// TIA Portal V20 export
DATA_BLOCK "CallUnit_DB"   // DB12
{ DB_Accessible_From_OPC_UA := 'FALSE' }
AUTHOR : ERsystem_FA2_DH. Kim
// stored: AssignedProDiagFB Unit1.ProDiag, DBAccessibleFromOPCUA false, DBAccessibleFromWebserver false, InstanceOfName Unit1.CallUnit, InstanceOfType FB, Namespace Unit1
"Unit1.CallUnit"
   // VAR_INPUT
   //    safetyReleased : Bool := TRUE;
   // END_VAR
   // VAR_OUTPUT
   //    acknowledgeSafety { ExternalWritable := 'False'} : Bool := FALSE;
   // END_VAR
   // VAR_IN_OUT
   //    globalStatus : "LAF_typeGeneralStatus";
   //    unitInterface : "LAF_typeUnitInterface";
   // END_VAR
   // VAR
   //    instManageAlarms { ExternalWritable := 'False'} : "LAF_ManageAlarms";
   //    instStatusCollector { ExternalWritable := 'False'} : "LUC_StatusCollector";
   //    instInterfaceManager { ExternalWritable := 'False'} : "LUC_InterfaceManager";
   //    instUnitModeStateManager { ExternalWritable := 'False'} : "LPMLV2022_UnitModeStateManager";
   //    instRemoteInterfaceOpcUa { ExternalWritable := 'False'} : "LUC_RemoteCtrl_OpcUa";
   //    instSignalStack { ExternalWritable := 'False'} : "LUC_SignalStack";
   //    instUnitModeStateTimes { ExternalWritable := 'False'} : "LPMLV2022_UnitModeStateTimes";
   //    instUnitModeChangeAllowed { ExternalWritable := 'False'} : "LPMLV2022_UnitModeChangeAllowed";
   //    instPFEEvents { S7_SetPoint := 'True'} : "Unit1.EventsPFE";
   //    statTonTime { S7_SetPoint := 'True'} : Array[0..99] of TON_TIME;
   //    instTofTimer { ExternalWritable := 'False'} : Array[0..9] of TOF_TIME;
   //    instEQP_Interface_BA010 { ExternalWritable := 'False'} : "LER_EQP_Interface_ReelCut";
   //    instEQP_Interface_BA015 { ExternalWritable := 'False'} : "LER_EQP_Interface_ReelCut";
   //    instEQP_Interface_BA060 { ExternalWritable := 'False'} : "LER_EQP_Interface_Inspection";
   //    instEQP_Interface_BA030 { ExternalWritable := 'False'} : "LER_EQP_Interface_OtherStack";
   //    BSEND_Instance_BA10 { S7_SetPoint := 'True'} : BSEND;
   //    BRCV_Instance_BA10 { S7_SetPoint := 'True'} : BRCV;
   //    BSEND_Instance_BA15 { S7_SetPoint := 'True'} : BSEND;
   //    BRCV_Instance_BA15 { S7_SetPoint := 'True'} : BRCV;
   //    BSEND_Instance_BA40 { S7_SetPoint := 'True'} : BSEND;
   //    BRCV_Instance_BA40 { S7_SetPoint := 'True'} : BRCV;
   //    BSEND_Instance_BA60 { S7_SetPoint := 'True'} : BSEND;
   //    BRCV_Instance_BA60 { S7_SetPoint := 'True'} : BRCV;
   //    instSinaInfeed { ExternalWritable := 'False'} : SinaInfeed;
   //    statRemoteInterface { ExternalWritable := 'False'} : "LUC_typeCommands";
   //    statLocalInterface { ExternalWritable := 'False'} : "LUC_typeCommands";
   //    statEmEnableCheck { ExternalWritable := 'False'} : Array[0..2] of Bool;
   //    statSpecialFuctionEnableCheck : Array[0..2] of Bool;
   //    statEmHomeScCheck { ExternalWritable := 'False'} : Array[0..7] of Bool;
   //    statPulse { ExternalWritable := 'False'} : Array[0..99] of Bool;
   //    statNoModeCmd { ExternalWritable := 'False'} : Bool;
   //    statEnableManualCmds : Bool;
   //    sleep { S7_SetPoint := 'True'} : "LER_typeSleepMode";
   //    statPreElectrodeNumber : Struct
   //       anode : DInt;
   //       cathode : DInt;
   //       currentTotalEL : DInt;
   //    END_STRUCT;
   //    instCalculateOut { S7_SetPoint := 'True'} : "LER_Calculate_Out";
   //    instStackMainCommand { S7_SetPoint := 'True'} : "LER_StackMainCommand";
   //    InstLER_FFU_LIU117 { S7_SetPoint := 'True'} : "LER_FFU_LIU117";
   //    sMotionToPLC { S7_SetPoint := 'True'} : "LER_typeCommonDataStackMotion";
   //    StatAllEmLinked { S7_SetPoint := 'True'} : Bool;
   //    citi_Ptrig : Array[0..20] of Bool;
   //    citiTon : Array[0..20] of TON_TIME;
   //    citi : Time;
   //    citiTest : Array[0..20] of Bool;
   //    statCalculateParameters : Struct
   //       AnodeCount : DInt;
   //       CathodeCount : DInt;
   //       SepaCount : DInt;
   //       TotalThickness : LReal;
   //       TotalSepaWebLenth : LReal;
   //    END_STRUCT;
   // END_VAR
BEGIN
   instManageAlarms.proDiagState.Total_Number := 562;
   instManageAlarms.proDiagState.All := FALSE;
   instManageAlarms.proDiagState.O := FALSE;
   instManageAlarms.proDiagState.I := FALSE;
   instManageAlarms.proDiagState.R := FALSE;
   instManageAlarms.proDiagState."A" := FALSE;
   instManageAlarms.proDiagState.P := FALSE;
   instManageAlarms.proDiagState.Merr := FALSE;
   instManageAlarms.proDiagState.Mtxt := FALSE;
   instManageAlarms.proDiagState.SV_Types := 16#00;
   instManageAlarms.proDiagState.C1 := FALSE;
   instManageAlarms.proDiagState.C2 := FALSE;
   instManageAlarms.proDiagState.C3 := FALSE;
   instManageAlarms.proDiagState.C4 := FALSE;
   instManageAlarms.proDiagState.C5 := FALSE;
   instManageAlarms.proDiagState.C6 := FALSE;
   instManageAlarms.proDiagState.C7 := FALSE;
   instManageAlarms.proDiagState.C8 := FALSE;
   instManageAlarms.proDiagState.Categories := 16#00;
   instManageAlarms.proDiagState.Sub_Cat_1 := 16#0000_0000;
   instManageAlarms.proDiagState.Sub_Cat_2 := 16#0000_0000;
   instManageAlarms.proDiagState.Reserved := 16#00;
   instManageAlarms.parentAlarmDB.error := FALSE;
   instManageAlarms.parentAlarmDB.warning := FALSE;
   instManageAlarms.parentAlarmDB.info := FALSE;
   instManageAlarms.alarmDB.error := FALSE;
   instManageAlarms.alarmDB.warning := FALSE;
   instManageAlarms.alarmDB.info := FALSE;
   instManageAlarms.hmiInterfaceDB.error := FALSE;
   instManageAlarms.hmiInterfaceDB.warning := FALSE;
   instManageAlarms.hmiInterfaceDB.info := FALSE;
   instInterfaceManager.processInterface.reset := FALSE;
   instInterfaceManager.processInterface.start := FALSE;
   instInterfaceManager.processInterface.stop := FALSE;
   instInterfaceManager.processInterface.hold := FALSE;
   instInterfaceManager.processInterface.unhold := FALSE;
   instInterfaceManager.processInterface.suspend := FALSE;
   instInterfaceManager.processInterface.unsuspend := FALSE;
   instInterfaceManager.processInterface.abort := FALSE;
   instInterfaceManager.processInterface.clear := FALSE;
   instInterfaceManager.processInterface.complete := FALSE;
   instInterfaceManager.processInterface.stateComplete := TRUE;
   instInterfaceManager.enableLocalInterface := TRUE;
   instInterfaceManager.localInterface.modeRequests.production := FALSE;
   instInterfaceManager.localInterface.modeRequests.maintenance := TRUE;
   instInterfaceManager.localInterface.modeRequests.manual := FALSE;
   instInterfaceManager.localInterface.modeRequests.nomode := FALSE;
   instInterfaceManager.localInterface.modeRequests.sleep := FALSE;
   instInterfaceManager.localInterface.modeRequests.deepsleep := FALSE;
   instInterfaceManager.localInterface.modeRequests.userMode04 := FALSE;
   instInterfaceManager.localInterface.modeRequests.userMode05 := FALSE;
   instInterfaceManager.localInterface.modeRequests.userMode06 := FALSE;
   instInterfaceManager.localInterface.modeRequests.userMode07 := FALSE;
   instInterfaceManager.localInterface.modeRequests.userMode08 := FALSE;
   instInterfaceManager.localInterface.modeRequests.userMode09 := FALSE;
   instInterfaceManager.localInterface.modeRequests.userMode10 := FALSE;
   instInterfaceManager.localInterface.modeRequests.userMode11 := FALSE;
   instInterfaceManager.localInterface.modeRequests.userMode12 := FALSE;
   instInterfaceManager.localInterface.modeRequests.userMode13 := FALSE;
   instInterfaceManager.localInterface.stateCommands.reset := FALSE;
   instInterfaceManager.localInterface.stateCommands.start := FALSE;
   instInterfaceManager.localInterface.stateCommands.stop := FALSE;
   instInterfaceManager.localInterface.stateCommands.hold := FALSE;
   instInterfaceManager.localInterface.stateCommands.unhold := FALSE;
   instInterfaceManager.localInterface.stateCommands.suspend := FALSE;
   instInterfaceManager.localInterface.stateCommands.unsuspend := FALSE;
   instInterfaceManager.localInterface.stateCommands.abort := FALSE;
   instInterfaceManager.localInterface.stateCommands.clear := FALSE;
   instInterfaceManager.localInterface.stateCommands.complete := FALSE;
   instInterfaceManager.localInterface.stateCommands.stateComplete := FALSE;
   instInterfaceManager.enableHmiInterface := FALSE;
   instInterfaceManager.hmiInterface.modeRequests.production := FALSE;
   instInterfaceManager.hmiInterface.modeRequests.maintenance := FALSE;
   instInterfaceManager.hmiInterface.modeRequests.manual := FALSE;
   instInterfaceManager.hmiInterface.modeRequests.nomode := FALSE;
   instInterfaceManager.hmiInterface.modeRequests.sleep := FALSE;
   instInterfaceManager.hmiInterface.modeRequests.deepsleep := FALSE;
   instInterfaceManager.hmiInterface.modeRequests.userMode04 := FALSE;
   instInterfaceManager.hmiInterface.modeRequests.userMode05 := FALSE;
   instInterfaceManager.hmiInterface.modeRequests.userMode06 := FALSE;
   instInterfaceManager.hmiInterface.modeRequests.userMode07 := FALSE;
   instInterfaceManager.hmiInterface.modeRequests.userMode08 := FALSE;
   instInterfaceManager.hmiInterface.modeRequests.userMode09 := FALSE;
   instInterfaceManager.hmiInterface.modeRequests.userMode10 := FALSE;
   instInterfaceManager.hmiInterface.modeRequests.userMode11 := FALSE;
   instInterfaceManager.hmiInterface.modeRequests.userMode12 := FALSE;
   instInterfaceManager.hmiInterface.modeRequests.userMode13 := FALSE;
   instInterfaceManager.hmiInterface.stateCommands.reset := FALSE;
   instInterfaceManager.hmiInterface.stateCommands.start := FALSE;
   instInterfaceManager.hmiInterface.stateCommands.stop := FALSE;
   instInterfaceManager.hmiInterface.stateCommands.hold := FALSE;
   instInterfaceManager.hmiInterface.stateCommands.unhold := FALSE;
   instInterfaceManager.hmiInterface.stateCommands.suspend := FALSE;
   instInterfaceManager.hmiInterface.stateCommands.unsuspend := FALSE;
   instInterfaceManager.hmiInterface.stateCommands.abort := FALSE;
   instInterfaceManager.hmiInterface.stateCommands.clear := FALSE;
   instInterfaceManager.hmiInterface.stateCommands.complete := FALSE;
   instInterfaceManager.hmiInterface.stateCommands.stateComplete := FALSE;
   instInterfaceManager.enableRemoteInterface := FALSE;
   instInterfaceManager.remoteInterface.modeRequests.production := FALSE;
   instInterfaceManager.remoteInterface.modeRequests.maintenance := FALSE;
   instInterfaceManager.remoteInterface.modeRequests.manual := FALSE;
   instInterfaceManager.remoteInterface.modeRequests.nomode := FALSE;
   instInterfaceManager.remoteInterface.modeRequests.sleep := FALSE;
   instInterfaceManager.remoteInterface.modeRequests.deepsleep := FALSE;
   instInterfaceManager.remoteInterface.modeRequests.userMode04 := FALSE;
   instInterfaceManager.remoteInterface.modeRequests.userMode05 := FALSE;
   instInterfaceManager.remoteInterface.modeRequests.userMode06 := FALSE;
   instInterfaceManager.remoteInterface.modeRequests.userMode07 := FALSE;
   instInterfaceManager.remoteInterface.modeRequests.userMode08 := FALSE;
   instInterfaceManager.remoteInterface.modeRequests.userMode09 := FALSE;
   instInterfaceManager.remoteInterface.modeRequests.userMode10 := FALSE;
   instInterfaceManager.remoteInterface.modeRequests.userMode11 := FALSE;
   instInterfaceManager.remoteInterface.modeRequests.userMode12 := FALSE;
   instInterfaceManager.remoteInterface.modeRequests.userMode13 := FALSE;
   instInterfaceManager.remoteInterface.stateCommands.reset := FALSE;
   instInterfaceManager.remoteInterface.stateCommands.start := FALSE;
   instInterfaceManager.remoteInterface.stateCommands.stop := FALSE;
   instInterfaceManager.remoteInterface.stateCommands.hold := FALSE;
   instInterfaceManager.remoteInterface.stateCommands.unhold := FALSE;
   instInterfaceManager.remoteInterface.stateCommands.suspend := FALSE;
   instInterfaceManager.remoteInterface.stateCommands.unsuspend := FALSE;
   instInterfaceManager.remoteInterface.stateCommands.abort := FALSE;
   instInterfaceManager.remoteInterface.stateCommands.clear := FALSE;
   instInterfaceManager.remoteInterface.stateCommands.complete := FALSE;
   instInterfaceManager.remoteInterface.stateCommands.stateComplete := FALSE;
   instInterfaceManager.unitMode := 0;
   instInterfaceManager.unitModeChangeRequest := FALSE;
   instInterfaceManager.cntrlCmd := 3;
   instInterfaceManager.cmdChangeRequest := FALSE;
   instInterfaceManager.SC := FALSE;
   instInterfaceManager.localControlEnabled := TRUE;
   instInterfaceManager.hmiControlEnabled := FALSE;
   instInterfaceManager.remoteControlEnabled := FALSE;
   instInterfaceManager.error := FALSE;
   instInterfaceManager.status := 16#0000;
   instInterfaceManager.statRequested.mode := 0;
   instInterfaceManager.statRequested.state := 0;
   instInterfaceManager.statPrevious.modesLocalInterface := 16#0002;
   instInterfaceManager.statPrevious.modesRemoteInterface := 16#0000;
   instInterfaceManager.statPrevious.modesHmiInterface := 16#0000;
   instInterfaceManager.statPrevious.statesProcessInterface := 16#0400;
   instInterfaceManager.statPrevious.statesLocalInterface := 16#0000;
   instInterfaceManager.statPrevious.statesRemoteInterface := 16#0000;
   instInterfaceManager.statPrevious.statesHmiInterface := 16#0000;
   instInterfaceManager.statStatus := 16#0000;
   instUnitModeStateManager.UnitMode := 0;
   instUnitModeStateManager.UnitModeChangeRequest := FALSE;
   instUnitModeStateManager.CntrlCmd := 3;
   instUnitModeStateManager.CmdChangeRequest := FALSE;
   instUnitModeStateManager.SC := FALSE;
   instUnitModeStateManager.configuration.EnabledModesCfg := 16#0000_001E;
   instUnitModeStateManager.configuration.DisabledStatesCfg[0..1] := 16#0000_0000;
   instUnitModeStateManager.configuration.DisabledStatesCfg[2] := 16#0003_6020;
   instUnitModeStateManager.configuration.DisabledStatesCfg[3] := 16#0003_7C28;
   instUnitModeStateManager.configuration.DisabledStatesCfg[4..16] := 16#0000_0000;
   instUnitModeStateManager.configuration.ModeTransitionCfg[0..16] := 16#0000_0214;
   instUnitModeStateManager.configuration.holdCmdCfg := 16#0000_0040;
   instUnitModeStateManager.configuration.completeCmdCfg := 16#0000_0860;
   instUnitModeStateManager.UnitModeCurrent := 2;
   instUnitModeStateManager.StateCurrent := 2;
   instUnitModeStateManager.StateRequested := 2;
   instUnitModeStateManager.StateChangeInProcess := FALSE;
   instUnitModeStateManager.CurDisabledStates := 16#0003_6020;
   instUnitModeStateManager.curHoldCmdCfg := 16#0000_0040;
   instUnitModeStateManager.curCompleteCmdCfg := 16#0000_0000;
   instUnitModeStateManager.unitModeChangeNotAllowed := FALSE;
   instUnitModeStateManager.cntrlCmdNotAllowed := FALSE;
   instUnitModeStateManager.diagnostics.bufferIndex := 7;
   instUnitModeStateManager.diagnostics.buffer[0].timestamp := DTL#2026-01-06-06:46:51.371465172;
   instUnitModeStateManager.diagnostics.buffer[1].timestamp := DTL#2026-01-06-06:46:51.374585015;
   instUnitModeStateManager.diagnostics.buffer[2].timestamp := DTL#2026-01-06-06:46:51.567016868;
   instUnitModeStateManager.diagnostics.buffer[3].timestamp := DTL#2026-01-06-06:46:55.878705971;
   instUnitModeStateManager.diagnostics.buffer[4].timestamp := DTL#2026-01-06-06:46:55.971592245;
   instUnitModeStateManager.diagnostics.buffer[5].timestamp := DTL#2026-01-06-06:46:58.882031211;
   instUnitModeStateManager.diagnostics.buffer[6].timestamp := DTL#2026-01-06-06:46:58.884831167;
   instUnitModeStateManager.diagnostics.buffer[7].timestamp := DTL#2026-01-06-06:46:58.887783077;
   instUnitModeStateManager.diagnostics.buffer[0..2].UnitModeCurrent := 2;
   instUnitModeStateManager.diagnostics.buffer[3..6].UnitModeCurrent := 4;
   instUnitModeStateManager.diagnostics.buffer[7].UnitModeCurrent := 2;
   instUnitModeStateManager.diagnostics.buffer[0].StateCurrent := 8;
   instUnitModeStateManager.diagnostics.buffer[1..3].StateCurrent := 9;
   instUnitModeStateManager.diagnostics.buffer[4..5].StateCurrent := 1;
   instUnitModeStateManager.diagnostics.buffer[6..7].StateCurrent := 2;
   instUnitModeStateManager.diagnostics.buffer[0].UnitMode := 0;
   instUnitModeStateManager.diagnostics.buffer[1].UnitMode := 2;
   instUnitModeStateManager.diagnostics.buffer[2].UnitMode := 4;
   instUnitModeStateManager.diagnostics.buffer[3..5].UnitMode := 0;
   instUnitModeStateManager.diagnostics.buffer[6].UnitMode := 2;
   instUnitModeStateManager.diagnostics.buffer[7].UnitMode := 0;
   instUnitModeStateManager.diagnostics.buffer[0..2].CntrlCmd := 8;
   instUnitModeStateManager.diagnostics.buffer[3].CntrlCmd := 9;
   instUnitModeStateManager.diagnostics.buffer[4..7].CntrlCmd := 3;
   instUnitModeStateManager.diagnostics.buffer[0].SC := TRUE;
   instUnitModeStateManager.diagnostics.buffer[1..4].SC := FALSE;
   instUnitModeStateManager.diagnostics.buffer[5].SC := TRUE;
   instUnitModeStateManager.diagnostics.buffer[6].SC := FALSE;
   instUnitModeStateManager.diagnostics.buffer[7].SC := TRUE;
   instUnitModeStateManager.diagnostics.buffer[0].message := 16#02;
   instUnitModeStateManager.diagnostics.buffer[1].message := 16#03;
   instUnitModeStateManager.diagnostics.buffer[2].message := 16#01;
   instUnitModeStateManager.diagnostics.buffer[3].message := 16#02;
   instUnitModeStateManager.diagnostics.buffer[4].message := 16#84;
   instUnitModeStateManager.diagnostics.buffer[5].message := 16#02;
   instUnitModeStateManager.diagnostics.buffer[6].message := 16#01;
   instUnitModeStateManager.diagnostics.buffer[7].message := 16#85;
   instUnitModeStateManager.statConfiguration.EnabledModesCfg := 16#0000_001E;
   instUnitModeStateManager.statConfiguration.DisabledStatesCfg[0..1] := 16#0000_0000;
   instUnitModeStateManager.statConfiguration.DisabledStatesCfg[2] := 16#0003_6020;
   instUnitModeStateManager.statConfiguration.DisabledStatesCfg[3] := 16#0003_7C28;
   instUnitModeStateManager.statConfiguration.DisabledStatesCfg[4] := 16#000FFFFF;
   instUnitModeStateManager.statConfiguration.DisabledStatesCfg[5..16] := 16#0000_0000;
   instUnitModeStateManager.statConfiguration.ModeTransitionCfg[0..16] := 16#0000_0214;
   instUnitModeStateManager.statConfiguration.holdCmdCfg := 16#0000_0040;
   instUnitModeStateManager.statConfiguration.completeCmdCfg := 16#0000_0860;
   instUnitModeStateManager.statUnitModeChangeRequest := FALSE;
   instUnitModeStateManager.statCmdChangeRequest := FALSE;
   instUnitModeStateManager.statFirstCycle := FALSE;
   instUnitModeStateManager.statSCOld := FALSE;
   instUnitModeStateManager.statUnitMode := 0;
   instUnitModeStateManager.statUnitModeOld := 0;
   instUnitModeStateManager.statUnitModeCurrentInternal := 2;
   instUnitModeStateManager.statUnitModeCurrentInternalOld := 0;
   instUnitModeStateManager.statStateCurrentOld := 2;
   instUnitModeStateManager.statStateInternal := 2;
   instUnitModeStateManager.statStateInternalOld := 0;
   instUnitModeStateManager.statCntrlCmdOld := 0;
   instUnitModeStateManager.statStatesInCurrentMode.clearing := TRUE;
   instUnitModeStateManager.statStatesInCurrentMode.stopped := TRUE;
   instUnitModeStateManager.statStatesInCurrentMode.starting := TRUE;
   instUnitModeStateManager.statStatesInCurrentMode.idle := TRUE;
   instUnitModeStateManager.statStatesInCurrentMode.suspended := FALSE;
   instUnitModeStateManager.statStatesInCurrentMode.execute := TRUE;
   instUnitModeStateManager.statStatesInCurrentMode.stopping := TRUE;
   instUnitModeStateManager.statStatesInCurrentMode.aborting := TRUE;
   instUnitModeStateManager.statStatesInCurrentMode.aborted := TRUE;
   instUnitModeStateManager.statStatesInCurrentMode.holding := TRUE;
   instUnitModeStateManager.statStatesInCurrentMode.held := TRUE;
   instUnitModeStateManager.statStatesInCurrentMode.unholding := TRUE;
   instUnitModeStateManager.statStatesInCurrentMode.suspending := FALSE;
   instUnitModeStateManager.statStatesInCurrentMode.unsuspending := FALSE;
   instUnitModeStateManager.statStatesInCurrentMode.resetting := TRUE;
   instUnitModeStateManager.statStatesInCurrentMode.completing := FALSE;
   instUnitModeStateManager.statStatesInCurrentMode.completed := FALSE;
   instUnitModeStateManager.statConsiderHoldCmdIn.starting := FALSE;
   instUnitModeStateManager.statConsiderHoldCmdIn.idle := FALSE;
   instUnitModeStateManager.statConsiderHoldCmdIn.suspended := FALSE;
   instUnitModeStateManager.statConsiderHoldCmdIn.execute := TRUE;
   instUnitModeStateManager.statConsiderHoldCmdIn.unholding := FALSE;
   instUnitModeStateManager.statConsiderHoldCmdIn.suspending := FALSE;
   instUnitModeStateManager.statConsiderHoldCmdIn.unsuspending := FALSE;
   instUnitModeStateManager.statConsiderHoldCmdIn.completing := FALSE;
   instUnitModeStateManager.statConsiderHoldCmdIn.completed := FALSE;
   instUnitModeStateManager.statConsiderCompleteCmdIn.suspended := FALSE;
   instUnitModeStateManager.statConsiderCompleteCmdIn.execute := FALSE;
   instUnitModeStateManager.statConsiderCompleteCmdIn.held := FALSE;
   instUnitModeStateManager.statCmdChangeRequestOld := FALSE;
   instUnitModeStateManager.statUnitModeChangeRequestOld := FALSE;
   instUnitModeStateManager.statDiagnosticsBufferIndex := 7;
   instUnitModeStateManager.statStateRequested := 2;
   instUnitModeStateManager.statUnitModeChangeNotAllowed := FALSE;
   instUnitModeStateManager.statCntrlCmdNotAllowed := FALSE;
   instRemoteInterfaceOpcUa.remoteControlEnabled := FALSE;
   instRemoteInterfaceOpcUa.currentState := 2;
   instRemoteInterfaceOpcUa.currentMode := 2;
   instRemoteInterfaceOpcUa.cntrlCmdDenied := FALSE;
   instRemoteInterfaceOpcUa.unitModeChangeNotAllowed := FALSE;
   instRemoteInterfaceOpcUa.configuration.enableMethods.reset := TRUE;
   instRemoteInterfaceOpcUa.configuration.enableMethods.start := TRUE;
   instRemoteInterfaceOpcUa.configuration.enableMethods.stop := TRUE;
   instRemoteInterfaceOpcUa.configuration.enableMethods.hold := TRUE;
   instRemoteInterfaceOpcUa.configuration.enableMethods.unhold := TRUE;
   instRemoteInterfaceOpcUa.configuration.enableMethods.suspend := TRUE;
   instRemoteInterfaceOpcUa.configuration.enableMethods.unsuspend := TRUE;
   instRemoteInterfaceOpcUa.configuration.enableMethods.abort := TRUE;
   instRemoteInterfaceOpcUa.configuration.enableMethods.clear := TRUE;
   instRemoteInterfaceOpcUa.configuration.enableMethods.complete := TRUE;
   instRemoteInterfaceOpcUa.configuration.enableMethods.stateComplete := TRUE;
   instRemoteInterfaceOpcUa.configuration.enableMethods.requestUnitMode := TRUE;
   instRemoteInterfaceOpcUa.configuration.enableMethods.requestUnitState := TRUE;
   instRemoteInterfaceOpcUa.error := FALSE;
   instRemoteInterfaceOpcUa.status := 16#0000;
   instRemoteInterfaceOpcUa.subfunctionStatus := 16#0000_0000;
   instRemoteInterfaceOpcUa.instReset.methodEnable := TRUE;
   instRemoteInterfaceOpcUa.instReset.remoteControlEnabled := FALSE;
   instRemoteInterfaceOpcUa.instReset.currentState := 2;
   instRemoteInterfaceOpcUa.instReset.cntrlCmdDenied := FALSE;
   instRemoteInterfaceOpcUa.instReset.error := FALSE;
   instRemoteInterfaceOpcUa.instReset.status := 16#7000;
   instRemoteInterfaceOpcUa.instReset.subfunctionStatus := 16#0000_0000;
   instRemoteInterfaceOpcUa.instReset.OPC_UA_ServerMethodPre_Instance.Done := FALSE;
   instRemoteInterfaceOpcUa.instReset.OPC_UA_ServerMethodPre_Instance.Busy := FALSE;
   instRemoteInterfaceOpcUa.instReset.OPC_UA_ServerMethodPre_Instance.Error := FALSE;
   instRemoteInterfaceOpcUa.instReset.OPC_UA_ServerMethodPre_Instance.Status := 16#0070_0000;
   instRemoteInterfaceOpcUa.instReset.OPC_UA_ServerMethodPre_Instance.UAMethod_Called := FALSE;
   instRemoteInterfaceOpcUa.instReset.OPC_UA_ServerMethodPost_Instance.UAMethod_Result := 16#0000_0000;
   instRemoteInterfaceOpcUa.instReset.OPC_UA_ServerMethodPost_Instance.UAMethod_Finished := FALSE;
   instRemoteInterfaceOpcUa.instReset.OPC_UA_ServerMethodPost_Instance.Done := FALSE;
   instRemoteInterfaceOpcUa.instReset.OPC_UA_ServerMethodPost_Instance.Busy := FALSE;
   instRemoteInterfaceOpcUa.instReset.OPC_UA_ServerMethodPost_Instance.Error := FALSE;
   instRemoteInterfaceOpcUa.instReset.OPC_UA_ServerMethodPost_Instance.Status := 16#0070_0000;
   instRemoteInterfaceOpcUa.instStart.methodEnable := TRUE;
   instRemoteInterfaceOpcUa.instStart.remoteControlEnabled := FALSE;
   instRemoteInterfaceOpcUa.instStart.currentState := 2;
   instRemoteInterfaceOpcUa.instStart.cntrlCmdDenied := FALSE;
   instRemoteInterfaceOpcUa.instStart.error := FALSE;
   instRemoteInterfaceOpcUa.instStart.status := 16#7000;
   instRemoteInterfaceOpcUa.instStart.subfunctionStatus := 16#0000_0000;
   instRemoteInterfaceOpcUa.instStart.OPC_UA_ServerMethodPre_Instance.Done := FALSE;
   instRemoteInterfaceOpcUa.instStart.OPC_UA_ServerMethodPre_Instance.Busy := FALSE;
   instRemoteInterfaceOpcUa.instStart.OPC_UA_ServerMethodPre_Instance.Error := FALSE;
   instRemoteInterfaceOpcUa.instStart.OPC_UA_ServerMethodPre_Instance.Status := 16#0070_0000;
   instRemoteInterfaceOpcUa.instStart.OPC_UA_ServerMethodPre_Instance.UAMethod_Called := FALSE;
   instRemoteInterfaceOpcUa.instStart.OPC_UA_ServerMethodPost_Instance.UAMethod_Result := 16#0000_0000;
   instRemoteInterfaceOpcUa.instStart.OPC_UA_ServerMethodPost_Instance.UAMethod_Finished := FALSE;
   instRemoteInterfaceOpcUa.instStart.OPC_UA_ServerMethodPost_Instance.Done := FALSE;
   instRemoteInterfaceOpcUa.instStart.OPC_UA_ServerMethodPost_Instance.Busy := FALSE;
   instRemoteInterfaceOpcUa.instStart.OPC_UA_ServerMethodPost_Instance.Error := FALSE;
   instRemoteInterfaceOpcUa.instStart.OPC_UA_ServerMethodPost_Instance.Status := 16#0070_0000;
   instRemoteInterfaceOpcUa.instStop.methodEnable := TRUE;
   instRemoteInterfaceOpcUa.instStop.remoteControlEnabled := FALSE;
   instRemoteInterfaceOpcUa.instStop.currentState := 2;
   instRemoteInterfaceOpcUa.instStop.cntrlCmdDenied := FALSE;
   instRemoteInterfaceOpcUa.instStop.error := FALSE;
   instRemoteInterfaceOpcUa.instStop.status := 16#7000;
   instRemoteInterfaceOpcUa.instStop.subfunctionStatus := 16#0000_0000;
   instRemoteInterfaceOpcUa.instStop.OPC_UA_ServerMethodPre_Instance.Done := FALSE;
   instRemoteInterfaceOpcUa.instStop.OPC_UA_ServerMethodPre_Instance.Busy := FALSE;
   instRemoteInterfaceOpcUa.instStop.OPC_UA_ServerMethodPre_Instance.Error := FALSE;
   instRemoteInterfaceOpcUa.instStop.OPC_UA_ServerMethodPre_Instance.Status := 16#0070_0000;
   instRemoteInterfaceOpcUa.instStop.OPC_UA_ServerMethodPre_Instance.UAMethod_Called := FALSE;
   instRemoteInterfaceOpcUa.instStop.OPC_UA_ServerMethodPost_Instance.UAMethod_Result := 16#0000_0000;
   instRemoteInterfaceOpcUa.instStop.OPC_UA_ServerMethodPost_Instance.UAMethod_Finished := FALSE;
   instRemoteInterfaceOpcUa.instStop.OPC_UA_ServerMethodPost_Instance.Done := FALSE;
   instRemoteInterfaceOpcUa.instStop.OPC_UA_ServerMethodPost_Instance.Busy := FALSE;
   instRemoteInterfaceOpcUa.instStop.OPC_UA_ServerMethodPost_Instance.Error := FALSE;
   instRemoteInterfaceOpcUa.instStop.OPC_UA_ServerMethodPost_Instance.Status := 16#0070_0000;
   instRemoteInterfaceOpcUa.instHold.methodEnable := TRUE;
   instRemoteInterfaceOpcUa.instHold.remoteControlEnabled := FALSE;
   instRemoteInterfaceOpcUa.instHold.currentState := 2;
   instRemoteInterfaceOpcUa.instHold.cntrlCmdDenied := FALSE;
   instRemoteInterfaceOpcUa.instHold.error := FALSE;
   instRemoteInterfaceOpcUa.instHold.status := 16#7000;
   instRemoteInterfaceOpcUa.instHold.subfunctionStatus := 16#0000_0000;
   instRemoteInterfaceOpcUa.instHold.OPC_UA_ServerMethodPre_Instance.Done := FALSE;
   instRemoteInterfaceOpcUa.instHold.OPC_UA_ServerMethodPre_Instance.Busy := FALSE;
   instRemoteInterfaceOpcUa.instHold.OPC_UA_ServerMethodPre_Instance.Error := FALSE;
   instRemoteInterfaceOpcUa.instHold.OPC_UA_ServerMethodPre_Instance.Status := 16#0070_0000;
   instRemoteInterfaceOpcUa.instHold.OPC_UA_ServerMethodPre_Instance.UAMethod_Called := FALSE;
   instRemoteInterfaceOpcUa.instHold.OPC_UA_ServerMethodPost_Instance.UAMethod_Result := 16#0000_0000;
   instRemoteInterfaceOpcUa.instHold.OPC_UA_ServerMethodPost_Instance.UAMethod_Finished := FALSE;
   instRemoteInterfaceOpcUa.instHold.OPC_UA_ServerMethodPost_Instance.Done := FALSE;
   instRemoteInterfaceOpcUa.instHold.OPC_UA_ServerMethodPost_Instance.Busy := FALSE;
   instRemoteInterfaceOpcUa.instHold.OPC_UA_ServerMethodPost_Instance.Error := FALSE;
   instRemoteInterfaceOpcUa.instHold.OPC_UA_ServerMethodPost_Instance.Status := 16#0070_0000;
   instRemoteInterfaceOpcUa.instUnhold.methodEnable := TRUE;
   instRemoteInterfaceOpcUa.instUnhold.remoteControlEnabled := FALSE;
   instRemoteInterfaceOpcUa.instUnhold.currentState := 2;
   instRemoteInterfaceOpcUa.instUnhold.cntrlCmdDenied := FALSE;
   instRemoteInterfaceOpcUa.instUnhold.error := FALSE;
   instRemoteInterfaceOpcUa.instUnhold.status := 16#7000;
   instRemoteInterfaceOpcUa.instUnhold.subfunctionStatus := 16#0000_0000;
   instRemoteInterfaceOpcUa.instUnhold.OPC_UA_ServerMethodPre_Instance.Done := FALSE;
   instRemoteInterfaceOpcUa.instUnhold.OPC_UA_ServerMethodPre_Instance.Busy := FALSE;
   instRemoteInterfaceOpcUa.instUnhold.OPC_UA_ServerMethodPre_Instance.Error := FALSE;
   instRemoteInterfaceOpcUa.instUnhold.OPC_UA_ServerMethodPre_Instance.Status := 16#0070_0000;
   instRemoteInterfaceOpcUa.instUnhold.OPC_UA_ServerMethodPre_Instance.UAMethod_Called := FALSE;
   instRemoteInterfaceOpcUa.instUnhold.OPC_UA_ServerMethodPost_Instance.UAMethod_Result := 16#0000_0000;
   instRemoteInterfaceOpcUa.instUnhold.OPC_UA_ServerMethodPost_Instance.UAMethod_Finished := FALSE;
   instRemoteInterfaceOpcUa.instUnhold.OPC_UA_ServerMethodPost_Instance.Done := FALSE;
   instRemoteInterfaceOpcUa.instUnhold.OPC_UA_ServerMethodPost_Instance.Busy := FALSE;
   instRemoteInterfaceOpcUa.instUnhold.OPC_UA_ServerMethodPost_Instance.Error := FALSE;
   instRemoteInterfaceOpcUa.instUnhold.OPC_UA_ServerMethodPost_Instance.Status := 16#0070_0000;
   instRemoteInterfaceOpcUa.instSuspend.methodEnable := TRUE;
   instRemoteInterfaceOpcUa.instSuspend.remoteControlEnabled := FALSE;
   instRemoteInterfaceOpcUa.instSuspend.currentState := 2;
   instRemoteInterfaceOpcUa.instSuspend.cntrlCmdDenied := FALSE;
   instRemoteInterfaceOpcUa.instSuspend.error := FALSE;
   instRemoteInterfaceOpcUa.instSuspend.status := 16#7000;
   instRemoteInterfaceOpcUa.instSuspend.subfunctionStatus := 16#0000_0000;
   instRemoteInterfaceOpcUa.instSuspend.OPC_UA_ServerMethodPre_Instance.Done := FALSE;
   instRemoteInterfaceOpcUa.instSuspend.OPC_UA_ServerMethodPre_Instance.Busy := FALSE;
   instRemoteInterfaceOpcUa.instSuspend.OPC_UA_ServerMethodPre_Instance.Error := FALSE;
   instRemoteInterfaceOpcUa.instSuspend.OPC_UA_ServerMethodPre_Instance.Status := 16#0070_0000;
   instRemoteInterfaceOpcUa.instSuspend.OPC_UA_ServerMethodPre_Instance.UAMethod_Called := FALSE;
   instRemoteInterfaceOpcUa.instSuspend.OPC_UA_ServerMethodPost_Instance.UAMethod_Result := 16#0000_0000;
   instRemoteInterfaceOpcUa.instSuspend.OPC_UA_ServerMethodPost_Instance.UAMethod_Finished := FALSE;
   instRemoteInterfaceOpcUa.instSuspend.OPC_UA_ServerMethodPost_Instance.Done := FALSE;
   instRemoteInterfaceOpcUa.instSuspend.OPC_UA_ServerMethodPost_Instance.Busy := FALSE;
   instRemoteInterfaceOpcUa.instSuspend.OPC_UA_ServerMethodPost_Instance.Error := FALSE;
   instRemoteInterfaceOpcUa.instSuspend.OPC_UA_ServerMethodPost_Instance.Status := 16#0070_0000;
   instRemoteInterfaceOpcUa.instUnsuspend.methodEnable := TRUE;
   instRemoteInterfaceOpcUa.instUnsuspend.remoteControlEnabled := FALSE;
   instRemoteInterfaceOpcUa.instUnsuspend.currentState := 2;
   instRemoteInterfaceOpcUa.instUnsuspend.cntrlCmdDenied := FALSE;
   instRemoteInterfaceOpcUa.instUnsuspend.error := FALSE;
   instRemoteInterfaceOpcUa.instUnsuspend.status := 16#7000;
   instRemoteInterfaceOpcUa.instUnsuspend.subfunctionStatus := 16#0000_0000;
   instRemoteInterfaceOpcUa.instUnsuspend.OPC_UA_ServerMethodPre_Instance.Done := FALSE;
   instRemoteInterfaceOpcUa.instUnsuspend.OPC_UA_ServerMethodPre_Instance.Busy := FALSE;
   instRemoteInterfaceOpcUa.instUnsuspend.OPC_UA_ServerMethodPre_Instance.Error := FALSE;
   instRemoteInterfaceOpcUa.instUnsuspend.OPC_UA_ServerMethodPre_Instance.Status := 16#0070_0000;
   instRemoteInterfaceOpcUa.instUnsuspend.OPC_UA_ServerMethodPre_Instance.UAMethod_Called := FALSE;
   instRemoteInterfaceOpcUa.instUnsuspend.OPC_UA_ServerMethodPost_Instance.UAMethod_Result := 16#0000_0000;
   instRemoteInterfaceOpcUa.instUnsuspend.OPC_UA_ServerMethodPost_Instance.UAMethod_Finished := FALSE;
   instRemoteInterfaceOpcUa.instUnsuspend.OPC_UA_ServerMethodPost_Instance.Done := FALSE;
   instRemoteInterfaceOpcUa.instUnsuspend.OPC_UA_ServerMethodPost_Instance.Busy := FALSE;
   instRemoteInterfaceOpcUa.instUnsuspend.OPC_UA_ServerMethodPost_Instance.Error := FALSE;
   instRemoteInterfaceOpcUa.instUnsuspend.OPC_UA_ServerMethodPost_Instance.Status := 16#0070_0000;
   instRemoteInterfaceOpcUa.instAbort.methodEnable := TRUE;
   instRemoteInterfaceOpcUa.instAbort.remoteControlEnabled := FALSE;
   instRemoteInterfaceOpcUa.instAbort.currentState := 2;
   instRemoteInterfaceOpcUa.instAbort.cntrlCmdDenied := FALSE;
   instRemoteInterfaceOpcUa.instAbort.error := FALSE;
   instRemoteInterfaceOpcUa.instAbort.status := 16#7000;
   instRemoteInterfaceOpcUa.instAbort.subfunctionStatus := 16#0000_0000;
   instRemoteInterfaceOpcUa.instAbort.OPC_UA_ServerMethodPre_Instance.Done := FALSE;
   instRemoteInterfaceOpcUa.instAbort.OPC_UA_ServerMethodPre_Instance.Busy := FALSE;
   instRemoteInterfaceOpcUa.instAbort.OPC_UA_ServerMethodPre_Instance.Error := FALSE;
   instRemoteInterfaceOpcUa.instAbort.OPC_UA_ServerMethodPre_Instance.Status := 16#0070_0000;
   instRemoteInterfaceOpcUa.instAbort.OPC_UA_ServerMethodPre_Instance.UAMethod_Called := FALSE;
   instRemoteInterfaceOpcUa.instAbort.OPC_UA_ServerMethodPost_Instance.UAMethod_Result := 16#0000_0000;
   instRemoteInterfaceOpcUa.instAbort.OPC_UA_ServerMethodPost_Instance.UAMethod_Finished := FALSE;
   instRemoteInterfaceOpcUa.instAbort.OPC_UA_ServerMethodPost_Instance.Done := FALSE;
   instRemoteInterfaceOpcUa.instAbort.OPC_UA_ServerMethodPost_Instance.Busy := FALSE;
   instRemoteInterfaceOpcUa.instAbort.OPC_UA_ServerMethodPost_Instance.Error := FALSE;
   instRemoteInterfaceOpcUa.instAbort.OPC_UA_ServerMethodPost_Instance.Status := 16#0070_0000;
   instRemoteInterfaceOpcUa.instClear.methodEnable := TRUE;
   instRemoteInterfaceOpcUa.instClear.remoteControlEnabled := FALSE;
   instRemoteInterfaceOpcUa.instClear.currentState := 2;
   instRemoteInterfaceOpcUa.instClear.cntrlCmdDenied := FALSE;
   instRemoteInterfaceOpcUa.instClear.error := FALSE;
   instRemoteInterfaceOpcUa.instClear.status := 16#7000;
   instRemoteInterfaceOpcUa.instClear.subfunctionStatus := 16#0000_0000;
   instRemoteInterfaceOpcUa.instClear.OPC_UA_ServerMethodPre_Instance.Done := FALSE;
   instRemoteInterfaceOpcUa.instClear.OPC_UA_ServerMethodPre_Instance.Busy := FALSE;
   instRemoteInterfaceOpcUa.instClear.OPC_UA_ServerMethodPre_Instance.Error := FALSE;
   instRemoteInterfaceOpcUa.instClear.OPC_UA_ServerMethodPre_Instance.Status := 16#0070_0000;
   instRemoteInterfaceOpcUa.instClear.OPC_UA_ServerMethodPre_Instance.UAMethod_Called := FALSE;
   instRemoteInterfaceOpcUa.instClear.OPC_UA_ServerMethodPost_Instance.UAMethod_Result := 16#0000_0000;
   instRemoteInterfaceOpcUa.instClear.OPC_UA_ServerMethodPost_Instance.UAMethod_Finished := FALSE;
   instRemoteInterfaceOpcUa.instClear.OPC_UA_ServerMethodPost_Instance.Done := FALSE;
   instRemoteInterfaceOpcUa.instClear.OPC_UA_ServerMethodPost_Instance.Busy := FALSE;
   instRemoteInterfaceOpcUa.instClear.OPC_UA_ServerMethodPost_Instance.Error := FALSE;
   instRemoteInterfaceOpcUa.instClear.OPC_UA_ServerMethodPost_Instance.Status := 16#0070_0000;
   instRemoteInterfaceOpcUa.instComplete.methodEnable := TRUE;
   instRemoteInterfaceOpcUa.instComplete.remoteControlEnabled := FALSE;
   instRemoteInterfaceOpcUa.instComplete.currentState := 2;
   instRemoteInterfaceOpcUa.instComplete.cntrlCmdDenied := FALSE;
   instRemoteInterfaceOpcUa.instComplete.error := FALSE;
   instRemoteInterfaceOpcUa.instComplete.status := 16#7000;
   instRemoteInterfaceOpcUa.instComplete.subfunctionStatus := 16#0000_0000;
   instRemoteInterfaceOpcUa.instComplete.OPC_UA_ServerMethodPre_Instance.Done := FALSE;
   instRemoteInterfaceOpcUa.instComplete.OPC_UA_ServerMethodPre_Instance.Busy := FALSE;
   instRemoteInterfaceOpcUa.instComplete.OPC_UA_ServerMethodPre_Instance.Error := FALSE;
   instRemoteInterfaceOpcUa.instComplete.OPC_UA_ServerMethodPre_Instance.Status := 16#0070_0000;
   instRemoteInterfaceOpcUa.instComplete.OPC_UA_ServerMethodPre_Instance.UAMethod_Called := FALSE;
   instRemoteInterfaceOpcUa.instComplete.OPC_UA_ServerMethodPost_Instance.UAMethod_Result := 16#0000_0000;
   instRemoteInterfaceOpcUa.instComplete.OPC_UA_ServerMethodPost_Instance.UAMethod_Finished := FALSE;
   instRemoteInterfaceOpcUa.instComplete.OPC_UA_ServerMethodPost_Instance.Done := FALSE;
   instRemoteInterfaceOpcUa.instComplete.OPC_UA_ServerMethodPost_Instance.Busy := FALSE;
   instRemoteInterfaceOpcUa.instComplete.OPC_UA_ServerMethodPost_Instance.Error := FALSE;
   instRemoteInterfaceOpcUa.instComplete.OPC_UA_ServerMethodPost_Instance.Status := 16#0070_0000;
   instRemoteInterfaceOpcUa.instStateComplete.methodEnable := TRUE;
   instRemoteInterfaceOpcUa.instStateComplete.remoteControlEnabled := FALSE;
   instRemoteInterfaceOpcUa.instStateComplete.currentState := 2;
   instRemoteInterfaceOpcUa.instStateComplete.cntrlCmdDenied := FALSE;
   instRemoteInterfaceOpcUa.instStateComplete.error := FALSE;
   instRemoteInterfaceOpcUa.instStateComplete.status := 16#7000;
   instRemoteInterfaceOpcUa.instStateComplete.subfunctionStatus := 16#0000_0000;
   instRemoteInterfaceOpcUa.instStateComplete.OPC_UA_ServerMethodPre_Instance.Done := FALSE;
   instRemoteInterfaceOpcUa.instStateComplete.OPC_UA_ServerMethodPre_Instance.Busy := FALSE;
   instRemoteInterfaceOpcUa.instStateComplete.OPC_UA_ServerMethodPre_Instance.Error := FALSE;
   instRemoteInterfaceOpcUa.instStateComplete.OPC_UA_ServerMethodPre_Instance.Status := 16#0070_0000;
   instRemoteInterfaceOpcUa.instStateComplete.OPC_UA_ServerMethodPre_Instance.UAMethod_Called := FALSE;
   instRemoteInterfaceOpcUa.instStateComplete.OPC_UA_ServerMethodPost_Instance.UAMethod_Result := 16#0000_0000;
   instRemoteInterfaceOpcUa.instStateComplete.OPC_UA_ServerMethodPost_Instance.UAMethod_Finished := FALSE;
   instRemoteInterfaceOpcUa.instStateComplete.OPC_UA_ServerMethodPost_Instance.Done := FALSE;
   instRemoteInterfaceOpcUa.instStateComplete.OPC_UA_ServerMethodPost_Instance.Busy := FALSE;
   instRemoteInterfaceOpcUa.instStateComplete.OPC_UA_ServerMethodPost_Instance.Error := FALSE;
   instRemoteInterfaceOpcUa.instStateComplete.OPC_UA_ServerMethodPost_Instance.Status := 16#0070_0000;
   instRemoteInterfaceOpcUa.instSetUnitMode.methodEnable := TRUE;
   instRemoteInterfaceOpcUa.instSetUnitMode.remoteControlEnabled := FALSE;
   instRemoteInterfaceOpcUa.instSetUnitMode.currentMode := 2;
   instRemoteInterfaceOpcUa.instSetUnitMode.unitModeChangeDenied := FALSE;
   instRemoteInterfaceOpcUa.instSetUnitMode.error := FALSE;
   instRemoteInterfaceOpcUa.instSetUnitMode.status := 16#7000;
   instRemoteInterfaceOpcUa.instSetUnitMode.subfunctionStatus := 16#0000_0000;
   instRemoteInterfaceOpcUa.instSetUnitMode.OPC_UA_ServerMethodPre_Instance.Done := FALSE;
   instRemoteInterfaceOpcUa.instSetUnitMode.OPC_UA_ServerMethodPre_Instance.Busy := FALSE;
   instRemoteInterfaceOpcUa.instSetUnitMode.OPC_UA_ServerMethodPre_Instance.Error := FALSE;
   instRemoteInterfaceOpcUa.instSetUnitMode.OPC_UA_ServerMethodPre_Instance.Status := 16#0070_0000;
   instRemoteInterfaceOpcUa.instSetUnitMode.OPC_UA_ServerMethodPre_Instance.UAMethod_Called := FALSE;
   instRemoteInterfaceOpcUa.instSetUnitMode.OPC_UA_ServerMethodPost_Instance.UAMethod_Result := 16#0000_0000;
   instRemoteInterfaceOpcUa.instSetUnitMode.OPC_UA_ServerMethodPost_Instance.UAMethod_Finished := FALSE;
   instRemoteInterfaceOpcUa.instSetUnitMode.OPC_UA_ServerMethodPost_Instance.Done := FALSE;
   instRemoteInterfaceOpcUa.instSetUnitMode.OPC_UA_ServerMethodPost_Instance.Busy := FALSE;
   instRemoteInterfaceOpcUa.instSetUnitMode.OPC_UA_ServerMethodPost_Instance.Error := FALSE;
   instRemoteInterfaceOpcUa.instSetUnitMode.OPC_UA_ServerMethodPost_Instance.Status := 16#0070_0000;
   instRemoteInterfaceOpcUa.instSetUnitMode.UAMethod_InParameters.RequestedMode := 0;
   instRemoteInterfaceOpcUa.instSetUnitMode.statLastCycleMode := 2;
   instRemoteInterfaceOpcUa.instSetUnitState.methodEnable := TRUE;
   instRemoteInterfaceOpcUa.instSetUnitState.remoteControlEnabled := FALSE;
   instRemoteInterfaceOpcUa.instSetUnitState.currentState := 2;
   instRemoteInterfaceOpcUa.instSetUnitState.cntrlCmdDenied := FALSE;
   instRemoteInterfaceOpcUa.instSetUnitState.error := FALSE;
   instRemoteInterfaceOpcUa.instSetUnitState.status := 16#7000;
   instRemoteInterfaceOpcUa.instSetUnitState.subfunctionStatus := 16#0000_0000;
   instRemoteInterfaceOpcUa.instSetUnitState.OPC_UA_ServerMethodPre_Instance.Done := FALSE;
   instRemoteInterfaceOpcUa.instSetUnitState.OPC_UA_ServerMethodPre_Instance.Busy := FALSE;
   instRemoteInterfaceOpcUa.instSetUnitState.OPC_UA_ServerMethodPre_Instance.Error := FALSE;
   instRemoteInterfaceOpcUa.instSetUnitState.OPC_UA_ServerMethodPre_Instance.Status := 16#0070_0000;
   instRemoteInterfaceOpcUa.instSetUnitState.OPC_UA_ServerMethodPre_Instance.UAMethod_Called := FALSE;
   instRemoteInterfaceOpcUa.instSetUnitState.OPC_UA_ServerMethodPost_Instance.UAMethod_Result := 16#0000_0000;
   instRemoteInterfaceOpcUa.instSetUnitState.OPC_UA_ServerMethodPost_Instance.UAMethod_Finished := FALSE;
   instRemoteInterfaceOpcUa.instSetUnitState.OPC_UA_ServerMethodPost_Instance.Done := FALSE;
   instRemoteInterfaceOpcUa.instSetUnitState.OPC_UA_ServerMethodPost_Instance.Busy := FALSE;
   instRemoteInterfaceOpcUa.instSetUnitState.OPC_UA_ServerMethodPost_Instance.Error := FALSE;
   instRemoteInterfaceOpcUa.instSetUnitState.OPC_UA_ServerMethodPost_Instance.Status := 16#0070_0000;
   instRemoteInterfaceOpcUa.instSetUnitState.UAMethod_InParameters.RequestedCommand := 0;
   instRemoteInterfaceOpcUa.instSetUnitState.statLastCycleState := 2;
   instSignalStack.currentState := 0;
   instSignalStack.freqClockBit := FALSE;
   instSignalStack.disableHorn := FALSE;
   instSignalStack.hornPulseTime := T#0MS;
   instSignalStack.processBypass.static.red := FALSE;
   instSignalStack.processBypass.static.yellow := FALSE;
   instSignalStack.processBypass.static.blue := FALSE;
   instSignalStack.processBypass.static.green := FALSE;
   instSignalStack.processBypass.static.horn := FALSE;
   instSignalStack.processBypass.static.white := FALSE;
   instSignalStack.processBypass.static.user1 := FALSE;
   instSignalStack.processBypass.static.user2 := FALSE;
   instSignalStack.processBypass.flashing.red := FALSE;
   instSignalStack.processBypass.flashing.yellow := FALSE;
   instSignalStack.processBypass.flashing.blue := FALSE;
   instSignalStack.processBypass.flashing.green := FALSE;
   instSignalStack.processBypass.flashing.horn := FALSE;
   instSignalStack.processBypass.flashing.white := FALSE;
   instSignalStack.processBypass.flashing.user1 := FALSE;
   instSignalStack.processBypass.flashing.user2 := FALSE;
   instSignalStack.configuration.undefined.static.red := FALSE;
   instSignalStack.configuration.undefined.static.yellow := FALSE;
   instSignalStack.configuration.undefined.static.blue := FALSE;
   instSignalStack.configuration.undefined.static.green := FALSE;
   instSignalStack.configuration.undefined.static.horn := FALSE;
   instSignalStack.configuration.undefined.static.white := FALSE;
   instSignalStack.configuration.undefined.static.user1 := FALSE;
   instSignalStack.configuration.undefined.static.user2 := FALSE;
   instSignalStack.configuration.undefined.flashing.red := TRUE;
   instSignalStack.configuration.undefined.flashing.yellow := FALSE;
   instSignalStack.configuration.undefined.flashing.blue := FALSE;
   instSignalStack.configuration.undefined.flashing.green := FALSE;
   instSignalStack.configuration.undefined.flashing.horn := FALSE;
   instSignalStack.configuration.undefined.flashing.white := FALSE;
   instSignalStack.configuration.undefined.flashing.user1 := FALSE;
   instSignalStack.configuration.undefined.flashing.user2 := FALSE;
   instSignalStack.configuration.clearing.static.red := FALSE;
   instSignalStack.configuration.clearing.static.yellow := FALSE;
   instSignalStack.configuration.clearing.static.blue := FALSE;
   instSignalStack.configuration.clearing.static.green := FALSE;
   instSignalStack.configuration.clearing.static.horn := FALSE;
   instSignalStack.configuration.clearing.static.white := FALSE;
   instSignalStack.configuration.clearing.static.user1 := FALSE;
   instSignalStack.configuration.clearing.static.user2 := FALSE;
   instSignalStack.configuration.clearing.flashing.red := TRUE;
   instSignalStack.configuration.clearing.flashing.yellow := FALSE;
   instSignalStack.configuration.clearing.flashing.blue := FALSE;
   instSignalStack.configuration.clearing.flashing.green := FALSE;
   instSignalStack.configuration.clearing.flashing.horn := FALSE;
   instSignalStack.configuration.clearing.flashing.white := FALSE;
   instSignalStack.configuration.clearing.flashing.user1 := FALSE;
   instSignalStack.configuration.clearing.flashing.user2 := FALSE;
   instSignalStack.configuration.stopped.static.red := TRUE;
   instSignalStack.configuration.stopped.static.yellow := FALSE;
   instSignalStack.configuration.stopped.static.blue := FALSE;
   instSignalStack.configuration.stopped.static.green := FALSE;
   instSignalStack.configuration.stopped.static.horn := FALSE;
   instSignalStack.configuration.stopped.static.white := FALSE;
   instSignalStack.configuration.stopped.static.user1 := FALSE;
   instSignalStack.configuration.stopped.static.user2 := FALSE;
   instSignalStack.configuration.stopped.flashing.red := FALSE;
   instSignalStack.configuration.stopped.flashing.yellow := FALSE;
   instSignalStack.configuration.stopped.flashing.blue := FALSE;
   instSignalStack.configuration.stopped.flashing.green := FALSE;
   instSignalStack.configuration.stopped.flashing.horn := FALSE;
   instSignalStack.configuration.stopped.flashing.white := FALSE;
   instSignalStack.configuration.stopped.flashing.user1 := FALSE;
   instSignalStack.configuration.stopped.flashing.user2 := FALSE;
   instSignalStack.configuration.starting.static.red := FALSE;
   instSignalStack.configuration.starting.static.yellow := FALSE;
   instSignalStack.configuration.starting.static.blue := FALSE;
   instSignalStack.configuration.starting.static.green := TRUE;
   instSignalStack.configuration.starting.static.horn := FALSE;
   instSignalStack.configuration.starting.static.white := FALSE;
   instSignalStack.configuration.starting.static.user1 := FALSE;
   instSignalStack.configuration.starting.static.user2 := FALSE;
   instSignalStack.configuration.starting.flashing.red := FALSE;
   instSignalStack.configuration.starting.flashing.yellow := FALSE;
   instSignalStack.configuration.starting.flashing.blue := FALSE;
   instSignalStack.configuration.starting.flashing.green := FALSE;
   instSignalStack.configuration.starting.flashing.horn := FALSE;
   instSignalStack.configuration.starting.flashing.white := FALSE;
   instSignalStack.configuration.starting.flashing.user1 := FALSE;
   instSignalStack.configuration.starting.flashing.user2 := FALSE;
   instSignalStack.configuration.idle.static.red := FALSE;
   instSignalStack.configuration.idle.static.yellow := FALSE;
   instSignalStack.configuration.idle.static.blue := FALSE;
   instSignalStack.configuration.idle.static.green := FALSE;
   instSignalStack.configuration.idle.static.horn := FALSE;
   instSignalStack.configuration.idle.static.white := FALSE;
   instSignalStack.configuration.idle.static.user1 := FALSE;
   instSignalStack.configuration.idle.static.user2 := FALSE;
   instSignalStack.configuration.idle.flashing.red := FALSE;
   instSignalStack.configuration.idle.flashing.yellow := FALSE;
   instSignalStack.configuration.idle.flashing.blue := FALSE;
   instSignalStack.configuration.idle.flashing.green := TRUE;
   instSignalStack.configuration.idle.flashing.horn := FALSE;
   instSignalStack.configuration.idle.flashing.white := FALSE;
   instSignalStack.configuration.idle.flashing.user1 := FALSE;
   instSignalStack.configuration.idle.flashing.user2 := FALSE;
   instSignalStack.configuration.suspended.static.red := FALSE;
   instSignalStack.configuration.suspended.static.yellow := TRUE;
   instSignalStack.configuration.suspended.static.blue := FALSE;
   instSignalStack.configuration.suspended.static.green := FALSE;
   instSignalStack.configuration.suspended.static.horn := FALSE;
   instSignalStack.configuration.suspended.static.white := FALSE;
   instSignalStack.configuration.suspended.static.user1 := FALSE;
   instSignalStack.configuration.suspended.static.user2 := FALSE;
   instSignalStack.configuration.suspended.flashing.red := FALSE;
   instSignalStack.configuration.suspended.flashing.yellow := FALSE;
   instSignalStack.configuration.suspended.flashing.blue := FALSE;
   instSignalStack.configuration.suspended.flashing.green := FALSE;
   instSignalStack.configuration.suspended.flashing.horn := FALSE;
   instSignalStack.configuration.suspended.flashing.white := FALSE;
   instSignalStack.configuration.suspended.flashing.user1 := FALSE;
   instSignalStack.configuration.suspended.flashing.user2 := FALSE;
   instSignalStack.configuration.execute.static.red := FALSE;
   instSignalStack.configuration.execute.static.yellow := FALSE;
   instSignalStack.configuration.execute.static.blue := FALSE;
   instSignalStack.configuration.execute.static.green := TRUE;
   instSignalStack.configuration.execute.static.horn := FALSE;
   instSignalStack.configuration.execute.static.white := FALSE;
   instSignalStack.configuration.execute.static.user1 := FALSE;
   instSignalStack.configuration.execute.static.user2 := FALSE;
   instSignalStack.configuration.execute.flashing.red := FALSE;
   instSignalStack.configuration.execute.flashing.yellow := FALSE;
   instSignalStack.configuration.execute.flashing.blue := FALSE;
   instSignalStack.configuration.execute.flashing.green := FALSE;
   instSignalStack.configuration.execute.flashing.horn := FALSE;
   instSignalStack.configuration.execute.flashing.white := FALSE;
   instSignalStack.configuration.execute.flashing.user1 := FALSE;
   instSignalStack.configuration.execute.flashing.user2 := FALSE;
   instSignalStack.configuration.stopping.static.red := TRUE;
   instSignalStack.configuration.stopping.static.yellow := FALSE;
   instSignalStack.configuration.stopping.static.blue := FALSE;
   instSignalStack.configuration.stopping.static.green := FALSE;
   instSignalStack.configuration.stopping.static.horn := FALSE;
   instSignalStack.configuration.stopping.static.white := FALSE;
   instSignalStack.configuration.stopping.static.user1 := FALSE;
   instSignalStack.configuration.stopping.static.user2 := FALSE;
   instSignalStack.configuration.stopping.flashing.red := FALSE;
   instSignalStack.configuration.stopping.flashing.yellow := FALSE;
   instSignalStack.configuration.stopping.flashing.blue := FALSE;
   instSignalStack.configuration.stopping.flashing.green := FALSE;
   instSignalStack.configuration.stopping.flashing.horn := FALSE;
   instSignalStack.configuration.stopping.flashing.white := FALSE;
   instSignalStack.configuration.stopping.flashing.user1 := FALSE;
   instSignalStack.configuration.stopping.flashing.user2 := FALSE;
   instSignalStack.configuration.aborting.static.red := FALSE;
   instSignalStack.configuration.aborting.static.yellow := FALSE;
   instSignalStack.configuration.aborting.static.blue := FALSE;
   instSignalStack.configuration.aborting.static.green := FALSE;
   instSignalStack.configuration.aborting.static.horn := FALSE;
   instSignalStack.configuration.aborting.static.white := FALSE;
   instSignalStack.configuration.aborting.static.user1 := FALSE;
   instSignalStack.configuration.aborting.static.user2 := FALSE;
   instSignalStack.configuration.aborting.flashing.red := TRUE;
   instSignalStack.configuration.aborting.flashing.yellow := FALSE;
   instSignalStack.configuration.aborting.flashing.blue := FALSE;
   instSignalStack.configuration.aborting.flashing.green := FALSE;
   instSignalStack.configuration.aborting.flashing.horn := FALSE;
   instSignalStack.configuration.aborting.flashing.white := FALSE;
   instSignalStack.configuration.aborting.flashing.user1 := FALSE;
   instSignalStack.configuration.aborting.flashing.user2 := FALSE;
   instSignalStack.configuration.aborted.static.red := FALSE;
   instSignalStack.configuration.aborted.static.yellow := FALSE;
   instSignalStack.configuration.aborted.static.blue := FALSE;
   instSignalStack.configuration.aborted.static.green := FALSE;
   instSignalStack.configuration.aborted.static.horn := FALSE;
   instSignalStack.configuration.aborted.static.white := FALSE;
   instSignalStack.configuration.aborted.static.user1 := FALSE;
   instSignalStack.configuration.aborted.static.user2 := FALSE;
   instSignalStack.configuration.aborted.flashing.red := TRUE;
   instSignalStack.configuration.aborted.flashing.yellow := FALSE;
   instSignalStack.configuration.aborted.flashing.blue := FALSE;
   instSignalStack.configuration.aborted.flashing.green := FALSE;
   instSignalStack.configuration.aborted.flashing.horn := FALSE;
   instSignalStack.configuration.aborted.flashing.white := FALSE;
   instSignalStack.configuration.aborted.flashing.user1 := FALSE;
   instSignalStack.configuration.aborted.flashing.user2 := FALSE;
   instSignalStack.configuration.holding.static.red := FALSE;
   instSignalStack.configuration.holding.static.yellow := FALSE;
   instSignalStack.configuration.holding.static.blue := FALSE;
   instSignalStack.configuration.holding.static.green := FALSE;
   instSignalStack.configuration.holding.static.horn := FALSE;
   instSignalStack.configuration.holding.static.white := FALSE;
   instSignalStack.configuration.holding.static.user1 := FALSE;
   instSignalStack.configuration.holding.static.user2 := FALSE;
   instSignalStack.configuration.holding.flashing.red := FALSE;
   instSignalStack.configuration.holding.flashing.yellow := FALSE;
   instSignalStack.configuration.holding.flashing.blue := TRUE;
   instSignalStack.configuration.holding.flashing.green := FALSE;
   instSignalStack.configuration.holding.flashing.horn := FALSE;
   instSignalStack.configuration.holding.flashing.white := FALSE;
   instSignalStack.configuration.holding.flashing.user1 := FALSE;
   instSignalStack.configuration.holding.flashing.user2 := FALSE;
   instSignalStack.configuration.held.static.red := FALSE;
   instSignalStack.configuration.held.static.yellow := FALSE;
   instSignalStack.configuration.held.static.blue := TRUE;
   instSignalStack.configuration.held.static.green := FALSE;
   instSignalStack.configuration.held.static.horn := FALSE;
   instSignalStack.configuration.held.static.white := FALSE;
   instSignalStack.configuration.held.static.user1 := FALSE;
   instSignalStack.configuration.held.static.user2 := FALSE;
   instSignalStack.configuration.held.flashing.red := FALSE;
   instSignalStack.configuration.held.flashing.yellow := FALSE;
   instSignalStack.configuration.held.flashing.blue := FALSE;
   instSignalStack.configuration.held.flashing.green := FALSE;
   instSignalStack.configuration.held.flashing.horn := FALSE;
   instSignalStack.configuration.held.flashing.white := FALSE;
   instSignalStack.configuration.held.flashing.user1 := FALSE;
   instSignalStack.configuration.held.flashing.user2 := FALSE;
   instSignalStack.configuration.unholding.static.red := FALSE;
   instSignalStack.configuration.unholding.static.yellow := FALSE;
   instSignalStack.configuration.unholding.static.blue := FALSE;
   instSignalStack.configuration.unholding.static.green := TRUE;
   instSignalStack.configuration.unholding.static.horn := FALSE;
   instSignalStack.configuration.unholding.static.white := FALSE;
   instSignalStack.configuration.unholding.static.user1 := FALSE;
   instSignalStack.configuration.unholding.static.user2 := FALSE;
   instSignalStack.configuration.unholding.flashing.red := FALSE;
   instSignalStack.configuration.unholding.flashing.yellow := FALSE;
   instSignalStack.configuration.unholding.flashing.blue := FALSE;
   instSignalStack.configuration.unholding.flashing.green := FALSE;
   instSignalStack.configuration.unholding.flashing.horn := FALSE;
   instSignalStack.configuration.unholding.flashing.white := FALSE;
   instSignalStack.configuration.unholding.flashing.user1 := FALSE;
   instSignalStack.configuration.unholding.flashing.user2 := FALSE;
   instSignalStack.configuration.suspending.static.red := FALSE;
   instSignalStack.configuration.suspending.static.yellow := FALSE;
   instSignalStack.configuration.suspending.static.blue := FALSE;
   instSignalStack.configuration.suspending.static.green := FALSE;
   instSignalStack.configuration.suspending.static.horn := FALSE;
   instSignalStack.configuration.suspending.static.white := FALSE;
   instSignalStack.configuration.suspending.static.user1 := FALSE;
   instSignalStack.configuration.suspending.static.user2 := FALSE;
   instSignalStack.configuration.suspending.flashing.red := FALSE;
   instSignalStack.configuration.suspending.flashing.yellow := TRUE;
   instSignalStack.configuration.suspending.flashing.blue := FALSE;
   instSignalStack.configuration.suspending.flashing.green := FALSE;
   instSignalStack.configuration.suspending.flashing.horn := FALSE;
   instSignalStack.configuration.suspending.flashing.white := FALSE;
   instSignalStack.configuration.suspending.flashing.user1 := FALSE;
   instSignalStack.configuration.suspending.flashing.user2 := FALSE;
   instSignalStack.configuration.unsuspending.static.red := FALSE;
   instSignalStack.configuration.unsuspending.static.yellow := FALSE;
   instSignalStack.configuration.unsuspending.static.blue := FALSE;
   instSignalStack.configuration.unsuspending.static.green := TRUE;
   instSignalStack.configuration.unsuspending.static.horn := FALSE;
   instSignalStack.configuration.unsuspending.static.white := FALSE;
   instSignalStack.configuration.unsuspending.static.user1 := FALSE;
   instSignalStack.configuration.unsuspending.static.user2 := FALSE;
   instSignalStack.configuration.unsuspending.flashing.red := FALSE;
   instSignalStack.configuration.unsuspending.flashing.yellow := FALSE;
   instSignalStack.configuration.unsuspending.flashing.blue := FALSE;
   instSignalStack.configuration.unsuspending.flashing.green := FALSE;
   instSignalStack.configuration.unsuspending.flashing.horn := FALSE;
   instSignalStack.configuration.unsuspending.flashing.white := FALSE;
   instSignalStack.configuration.unsuspending.flashing.user1 := FALSE;
   instSignalStack.configuration.unsuspending.flashing.user2 := FALSE;
   instSignalStack.configuration.resetting.static.red := TRUE;
   instSignalStack.configuration.resetting.static.yellow := FALSE;
   instSignalStack.configuration.resetting.static.blue := FALSE;
   instSignalStack.configuration.resetting.static.green := FALSE;
   instSignalStack.configuration.resetting.static.horn := FALSE;
   instSignalStack.configuration.resetting.static.white := FALSE;
   instSignalStack.configuration.resetting.static.user1 := FALSE;
   instSignalStack.configuration.resetting.static.user2 := FALSE;
   instSignalStack.configuration.resetting.flashing.red := FALSE;
   instSignalStack.configuration.resetting.flashing.yellow := FALSE;
   instSignalStack.configuration.resetting.flashing.blue := FALSE;
   instSignalStack.configuration.resetting.flashing.green := FALSE;
   instSignalStack.configuration.resetting.flashing.horn := FALSE;
   instSignalStack.configuration.resetting.flashing.white := FALSE;
   instSignalStack.configuration.resetting.flashing.user1 := FALSE;
   instSignalStack.configuration.resetting.flashing.user2 := FALSE;
   instSignalStack.configuration.completing.static.red := FALSE;
   instSignalStack.configuration.completing.static.yellow := FALSE;
   instSignalStack.configuration.completing.static.blue := FALSE;
   instSignalStack.configuration.completing.static.green := TRUE;
   instSignalStack.configuration.completing.static.horn := FALSE;
   instSignalStack.configuration.completing.static.white := FALSE;
   instSignalStack.configuration.completing.static.user1 := FALSE;
   instSignalStack.configuration.completing.static.user2 := FALSE;
   instSignalStack.configuration.completing.flashing.red := FALSE;
   instSignalStack.configuration.completing.flashing.yellow := FALSE;
   instSignalStack.configuration.completing.flashing.blue := FALSE;
   instSignalStack.configuration.completing.flashing.green := FALSE;
   instSignalStack.configuration.completing.flashing.horn := FALSE;
   instSignalStack.configuration.completing.flashing.white := FALSE;
   instSignalStack.configuration.completing.flashing.user1 := FALSE;
   instSignalStack.configuration.completing.flashing.user2 := FALSE;
   instSignalStack.configuration.completed.static.red := TRUE;
   instSignalStack.configuration.completed.static.yellow := FALSE;
   instSignalStack.configuration.completed.static.blue := FALSE;
   instSignalStack.configuration.completed.static.green := FALSE;
   instSignalStack.configuration.completed.static.horn := FALSE;
   instSignalStack.configuration.completed.static.white := FALSE;
   instSignalStack.configuration.completed.static.user1 := FALSE;
   instSignalStack.configuration.completed.static.user2 := FALSE;
   instSignalStack.configuration.completed.flashing.red := FALSE;
   instSignalStack.configuration.completed.flashing.yellow := FALSE;
   instSignalStack.configuration.completed.flashing.blue := FALSE;
   instSignalStack.configuration.completed.flashing.green := FALSE;
   instSignalStack.configuration.completed.flashing.horn := FALSE;
   instSignalStack.configuration.completed.flashing.white := FALSE;
   instSignalStack.configuration.completed.flashing.user1 := FALSE;
   instSignalStack.configuration.completed.flashing.user2 := FALSE;
   instSignalStack.lightsByBool.redSolid := FALSE;
   instSignalStack.lightsByBool.redFlashing := FALSE;
   instSignalStack.lightsByBool.yellowSolid := FALSE;
   instSignalStack.lightsByBool.yellowFlashing := FALSE;
   instSignalStack.lightsByBool.blueSolid := FALSE;
   instSignalStack.lightsByBool.blueFlashing := FALSE;
   instSignalStack.lightsByBool.greenSolid := FALSE;
   instSignalStack.lightsByBool.greenFlashing := FALSE;
   instSignalStack.lightsByBool.hornSolid := FALSE;
   instSignalStack.lightsByBool.hornFlashing := FALSE;
   instSignalStack.lightsByBool.whiteSolid := FALSE;
   instSignalStack.lightsByBool.whiteFlashing := FALSE;
   instSignalStack.lightsByBool.user1Solid := FALSE;
   instSignalStack.lightsByBool.user1Flashing := FALSE;
   instSignalStack.lightsByBool.user2Solid := FALSE;
   instSignalStack.lightsByBool.user2Flashing := FALSE;
   instSignalStack.lightsByDint.red := 0;
   instSignalStack.lightsByDint.yellow := 0;
   instSignalStack.lightsByDint.blue := 0;
   instSignalStack.lightsByDint.green := 0;
   instSignalStack.lightsByDint.horn := 0;
   instSignalStack.lightsByDint.white := 0;
   instSignalStack.lightsByDint.user1 := 0;
   instSignalStack.lightsByDint.user2 := 0;
   instSignalStack.lightsByDWord.statusByDWord := 16#0000_0000;
   instSignalStack.lightsStatus.red := FALSE;
   instSignalStack.lightsStatus.yellow := FALSE;
   instSignalStack.lightsStatus.blue := FALSE;
   instSignalStack.lightsStatus.green := FALSE;
   instSignalStack.lightsStatus.horn := FALSE;
   instSignalStack.lightsStatus.white := FALSE;
   instSignalStack.lightsStatus.user1 := FALSE;
   instSignalStack.lightsStatus.user2 := FALSE;
   instSignalStack.instPulseHorn.PT := T#1S;
   instSignalStack.instPulseHorn.IN := FALSE;
   instUnitModeStateTimes.UnitModeCurrent := 2;
   instUnitModeStateTimes.StateCurrent := 2;
   instUnitModeStateTimes.resetTimes := FALSE;
   instUnitModeStateTimes.ModeTimeCurrent := 47401;
   instUnitModeStateTimes.StateTimeCurrent := 47401;
   instUnitModeStateTimes.AccTimeSinceReset := 71237;
   instUnitModeStateTimes.actualTimeAllModes[0..1] := 0;
   instUnitModeStateTimes.actualTimeAllModes[2] := 47401;
   instUnitModeStateTimes.actualTimeAllModes[3] := 0;
   instUnitModeStateTimes.actualTimeAllModes[4] := 8;
   instUnitModeStateTimes.actualTimeAllModes[5..16] := 0;
   instUnitModeStateTimes.cumulativeTimeAllModes[0..1] := 0;
   instUnitModeStateTimes.cumulativeTimeAllModes[2] := 67801;
   instUnitModeStateTimes.cumulativeTimeAllModes[3] := 0;
   instUnitModeStateTimes.cumulativeTimeAllModes[4] := 3436;
   instUnitModeStateTimes.cumulativeTimeAllModes[5..16] := 0;
   instUnitModeStateTimes.actualTimeAllStatesOfAllModes[0,0..17] := 0;
   instUnitModeStateTimes.actualTimeAllStatesOfAllModes[1,0..17] := 0;
   instUnitModeStateTimes.actualTimeAllStatesOfAllModes[2,0] := 0;
   instUnitModeStateTimes.actualTimeAllStatesOfAllModes[2,1] := 3;
   instUnitModeStateTimes.actualTimeAllStatesOfAllModes[2,2] := 47401;
   instUnitModeStateTimes.actualTimeAllStatesOfAllModes[2,3..17] := 0;
   instUnitModeStateTimes.actualTimeAllStatesOfAllModes[3,0..17] := 0;
   instUnitModeStateTimes.actualTimeAllStatesOfAllModes[4,0] := 0;
   instUnitModeStateTimes.actualTimeAllStatesOfAllModes[4,1] := 3;
   instUnitModeStateTimes.actualTimeAllStatesOfAllModes[4,2..8] := 0;
   instUnitModeStateTimes.actualTimeAllStatesOfAllModes[4,9] := 5;
   instUnitModeStateTimes.actualTimeAllStatesOfAllModes[4,10..17] := 0;
   instUnitModeStateTimes.actualTimeAllStatesOfAllModes[5,0..17] := 0;
   instUnitModeStateTimes.actualTimeAllStatesOfAllModes[6,0..17] := 0;
   instUnitModeStateTimes.actualTimeAllStatesOfAllModes[7,0..17] := 0;
   instUnitModeStateTimes.actualTimeAllStatesOfAllModes[8,0..17] := 0;
   instUnitModeStateTimes.actualTimeAllStatesOfAllModes[9,0..17] := 0;
   instUnitModeStateTimes.actualTimeAllStatesOfAllModes[10,0..17] := 0;
   instUnitModeStateTimes.actualTimeAllStatesOfAllModes[11,0..17] := 0;
   instUnitModeStateTimes.actualTimeAllStatesOfAllModes[12,0..17] := 0;
   instUnitModeStateTimes.actualTimeAllStatesOfAllModes[13,0..17] := 0;
   instUnitModeStateTimes.actualTimeAllStatesOfAllModes[14,0..17] := 0;
   instUnitModeStateTimes.actualTimeAllStatesOfAllModes[15,0..17] := 0;
   instUnitModeStateTimes.actualTimeAllStatesOfAllModes[16,0..17] := 0;
   instUnitModeStateTimes.cumulativeTimeAllStatesOfAllModes[0,0..17] := 0;
   instUnitModeStateTimes.cumulativeTimeAllStatesOfAllModes[1,0..17] := 0;
   instUnitModeStateTimes.cumulativeTimeAllStatesOfAllModes[2,0] := 0;
   instUnitModeStateTimes.cumulativeTimeAllStatesOfAllModes[2,1] := 29;
   instUnitModeStateTimes.cumulativeTimeAllStatesOfAllModes[2,2] := 62920;
   instUnitModeStateTimes.cumulativeTimeAllStatesOfAllModes[2,3..7] := 0;
   instUnitModeStateTimes.cumulativeTimeAllStatesOfAllModes[2,8] := 1;
   instUnitModeStateTimes.cumulativeTimeAllStatesOfAllModes[2,9] := 4851;
   instUnitModeStateTimes.cumulativeTimeAllStatesOfAllModes[2,10..17] := 0;
   instUnitModeStateTimes.cumulativeTimeAllStatesOfAllModes[3,0..17] := 0;
   instUnitModeStateTimes.cumulativeTimeAllStatesOfAllModes[4,0] := 0;
   instUnitModeStateTimes.cumulativeTimeAllStatesOfAllModes[4,1] := 35;
   instUnitModeStateTimes.cumulativeTimeAllStatesOfAllModes[4,2..8] := 0;
   instUnitModeStateTimes.cumulativeTimeAllStatesOfAllModes[4,9] := 3401;
   instUnitModeStateTimes.cumulativeTimeAllStatesOfAllModes[4,10..17] := 0;
   instUnitModeStateTimes.cumulativeTimeAllStatesOfAllModes[5,0..17] := 0;
   instUnitModeStateTimes.cumulativeTimeAllStatesOfAllModes[6,0..17] := 0;
   instUnitModeStateTimes.cumulativeTimeAllStatesOfAllModes[7,0..17] := 0;
   instUnitModeStateTimes.cumulativeTimeAllStatesOfAllModes[8,0..17] := 0;
   instUnitModeStateTimes.cumulativeTimeAllStatesOfAllModes[9,0..17] := 0;
   instUnitModeStateTimes.cumulativeTimeAllStatesOfAllModes[10,0..17] := 0;
   instUnitModeStateTimes.cumulativeTimeAllStatesOfAllModes[11,0..17] := 0;
   instUnitModeStateTimes.cumulativeTimeAllStatesOfAllModes[12,0..17] := 0;
   instUnitModeStateTimes.cumulativeTimeAllStatesOfAllModes[13,0..17] := 0;
   instUnitModeStateTimes.cumulativeTimeAllStatesOfAllModes[14,0..17] := 0;
   instUnitModeStateTimes.cumulativeTimeAllStatesOfAllModes[15,0..17] := 0;
   instUnitModeStateTimes.cumulativeTimeAllStatesOfAllModes[16,0..17] := 0;
   instUnitModeStateTimes.actualTimeAllStatesOfCurrentMode[0] := 0;
   instUnitModeStateTimes.actualTimeAllStatesOfCurrentMode[1] := 3;
   instUnitModeStateTimes.actualTimeAllStatesOfCurrentMode[2] := 47401;
   instUnitModeStateTimes.actualTimeAllStatesOfCurrentMode[3..17] := 0;
   instUnitModeStateTimes.cumulativeTimeAllStatesOfCurrentMode[0] := 0;
   instUnitModeStateTimes.cumulativeTimeAllStatesOfCurrentMode[1] := 29;
   instUnitModeStateTimes.cumulativeTimeAllStatesOfCurrentMode[2] := 62920;
   instUnitModeStateTimes.cumulativeTimeAllStatesOfCurrentMode[3..7] := 0;
   instUnitModeStateTimes.cumulativeTimeAllStatesOfCurrentMode[8] := 1;
   instUnitModeStateTimes.cumulativeTimeAllStatesOfCurrentMode[9] := 4851;
   instUnitModeStateTimes.cumulativeTimeAllStatesOfCurrentMode[10..17] := 0;
   instUnitModeStateTimes.cumulativeTimeCurrentMode := 67801;
   instUnitModeStateTimes.statUnitModeCurrentOld := 2;
   instUnitModeStateTimes.statStateCurrentOld := 2;
   instUnitModeStateTimes.statResetTimesOld := FALSE;
   instUnitModeStateTimes.statStartingPointMeasureRuntime := 2.78082814701851E-308;
   instUnitModeStateTimes.statRuntime := 0.714137883731914;
   instUnitModeStateTimes.statFirstCycle := FALSE;
   instUnitModeStateTimes.statCurrentModeCurrentTime := 47401;
   instUnitModeStateTimes.statCurrentStateCurrentTime := 47401;
   statTonTime[0].PT := T#0MS;
   statTonTime[1].PT := T#1S;
   statTonTime[2..99].PT := T#0MS;
   statTonTime[0..99].IN := FALSE;
   statRemoteInterface.modeRequests.production := FALSE;
   statRemoteInterface.modeRequests.maintenance := FALSE;
   statRemoteInterface.modeRequests.manual := FALSE;
   statRemoteInterface.modeRequests.nomode := FALSE;
   statRemoteInterface.modeRequests.sleep := FALSE;
   statRemoteInterface.modeRequests.deepsleep := FALSE;
   statRemoteInterface.modeRequests.userMode04 := FALSE;
   statRemoteInterface.modeRequests.userMode05 := FALSE;
   statRemoteInterface.modeRequests.userMode06 := FALSE;
   statRemoteInterface.modeRequests.userMode07 := FALSE;
   statRemoteInterface.modeRequests.userMode08 := FALSE;
   statRemoteInterface.modeRequests.userMode09 := FALSE;
   statRemoteInterface.modeRequests.userMode10 := FALSE;
   statRemoteInterface.modeRequests.userMode11 := FALSE;
   statRemoteInterface.modeRequests.userMode12 := FALSE;
   statRemoteInterface.modeRequests.userMode13 := FALSE;
   statRemoteInterface.stateCommands.reset := FALSE;
   statRemoteInterface.stateCommands.start := FALSE;
   statRemoteInterface.stateCommands.stop := FALSE;
   statRemoteInterface.stateCommands.hold := FALSE;
   statRemoteInterface.stateCommands.unhold := FALSE;
   statRemoteInterface.stateCommands.suspend := FALSE;
   statRemoteInterface.stateCommands.unsuspend := FALSE;
   statRemoteInterface.stateCommands.abort := FALSE;
   statRemoteInterface.stateCommands.clear := FALSE;
   statRemoteInterface.stateCommands.complete := FALSE;
   statRemoteInterface.stateCommands.stateComplete := FALSE;
   statLocalInterface.modeRequests.production := FALSE;
   statLocalInterface.modeRequests.maintenance := TRUE;
   statLocalInterface.modeRequests.manual := FALSE;
   statLocalInterface.modeRequests.nomode := FALSE;
   statLocalInterface.modeRequests.sleep := FALSE;
   statLocalInterface.modeRequests.deepsleep := FALSE;
   statLocalInterface.modeRequests.userMode04 := FALSE;
   statLocalInterface.modeRequests.userMode05 := FALSE;
   statLocalInterface.modeRequests.userMode06 := FALSE;
   statLocalInterface.modeRequests.userMode07 := FALSE;
   statLocalInterface.modeRequests.userMode08 := FALSE;
   statLocalInterface.modeRequests.userMode09 := FALSE;
   statLocalInterface.modeRequests.userMode10 := FALSE;
   statLocalInterface.modeRequests.userMode11 := FALSE;
   statLocalInterface.modeRequests.userMode12 := FALSE;
   statLocalInterface.modeRequests.userMode13 := FALSE;
   statLocalInterface.stateCommands.reset := FALSE;
   statLocalInterface.stateCommands.start := FALSE;
   statLocalInterface.stateCommands.stop := FALSE;
   statLocalInterface.stateCommands.hold := FALSE;
   statLocalInterface.stateCommands.unhold := FALSE;
   statLocalInterface.stateCommands.suspend := FALSE;
   statLocalInterface.stateCommands.unsuspend := FALSE;
   statLocalInterface.stateCommands.abort := FALSE;
   statLocalInterface.stateCommands.clear := FALSE;
   statLocalInterface.stateCommands.complete := FALSE;
   statLocalInterface.stateCommands.stateComplete := FALSE;
END_DATA_BLOCK
